FUNCTION F_GetRampUpTimeString : STRING
VAR_INPUT
	fTargetTemp	: LREAL;
	fRampRate	: LREAL; 
	fCurrentTemp: LREAL;
END_VAR
VAR
	fFractionalTime		: LREAL;
	dwFractionalTime	: DWORD;
	tFractionalTime		: TIME;
	sFractionalTime		: STRING;
	
	mCharIndex	: INT;
	iHours		: INT;
	iMinutes	: INT;
	strFractionalTimeString	: STRING;
	strTrimmedTimeString	: STRING;
END_VAR

(*
// Calculate time in Hours
IF(stPlatform.stTestController.stOutputs.eTestState = E_TestStates.eTS_RampUp) THEN
	fFractionalTime := ((fTargetTemp - fCurrentTemp) / fRampRate) + stPlatform.stTestController.stInputs.fSoakTime;
ELSE
	fFractionalTime := stPlatform.stTestController.stInputs.fSoakTime - (stPlatform.stTestController.stInternal.fSoakTimer / 3600);
END_IF
// Convert time to ms 
fFractionalTime	:= fFractionalTime * 3.6E6;

// Convert to DW 
dwFractionalTime	:= LREAL_TO_DWORD(fFractionalTime);

// Convert to time
tFractionalTime		:= DWORD_TO_TIME(dwFractionalTime);

// Convert to string 
strFractionalTimeString := TIME_TO_STRING(tFractionalTime);

mCharIndex	:= FIND(STR2:= 'm',STR1:= strFractionalTimeString);
strTrimmedTimeString	:= LEFT(STR:=strFractionalTimeString,SIZE:=mCharIndex);

//strFractionalTimeString	:= LREAL_TO_STRING(fFractionalTime);

//F_GetRampUpTimeString	:= CONCAT(STR1:='Machine is Ramping Up. Load application required in  ',STR2:= CONCAT(STR1:= INT_TO_STRING(iHours), STR2:= (CONCAT(STR1:= ' Hours and ', STR2:=(CONCAT(STR1:= INT_TO_STRING(iMinutes),STR2:= ' Minutes.'))))));

F_GetRampUpTimeString	:= CONCAT(STR1:='Machine is Ramping Up. Load application required in  ',STR2:= strTrimmedTimeString);

*)

END_FUNCTION

(* stored: Version 1.1.0.1, ProductVersion 3.1.4024.12
   POU F_GetRampUpTimeString: Id {475f6d4a-fe2b-448e-a7de-c4ba9dd1eae2}, SpecialFunc None *)
